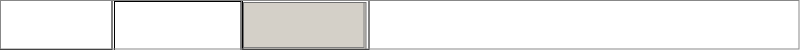
VISUALIZATION Nav  // 800x50
    Rectangle (-15,0 127x50)
    Rectangle (114,1 127x50)
    Rectangle (242,0 127x50)
    Button (243,2 123x47)
        OnMouseDown: change screen: Visualization
END_VISUALIZATION

(* stored: Version 1.1.0.1, ProductVersion 3.1.4024.12
   Visu Nav: Id {656f78cb-40bb-42de-86c9-a5ed5c4bf959} *)
